(* CODESYS project Magazijn Structured Tekst 2V0 - Opdracht 3.project
   Company: Avans
   Description: Simulatie voor opstelling Sorteer Station.
   Title: Simulatie Sorteer Station
   Author: Rene Potters/Gerard Harkema
   Version: 0.1.0

Project tree, tasks and I/O mapping:
  Device : CODESYS Control Win V3, 3S - Smart Software Solutions GmbH, version 3.5.13.20
    application MagazijnOverzetterStation
      libraries: Standard, * (System); Util, * (System); VisuDialogs, 3.5.12.0 (System)
      task MainTask (cyclic, interval t#20ms, priority 1) calls Main
      task Simulatie (cyclic, interval t#20ms, priority 1) calls OverzetterSim, MagazijnSim
    application MagazijnTest
      libraries: Standard, * (System); Util, * (System); VisuDialogs, 3.5.12.0 (System)
      task MainTask (cyclic, interval t#20ms, priority 1) calls MagazijnTest
      task Simulatie (cyclic, interval t#20ms, priority 1) calls MagazijnSim
    application OverzetterTest
      libraries: Standard, * (System); Util, * (System); VisuDialogs, 3.5.12.0 (System)
      task MainTask (cyclic, interval t#20ms, priority 1) calls OverzetterTest
      task Simulatie (cyclic, interval t#20ms, priority 1) calls OverzetterSim
  Simulatie/
    program MagazijnSim [ST]
    global variables SIM
    program OverzetterSim [ST]
    data type OverzetterDUT
    data type MagazijnDUT
  text list GlobalTextList
  Programma Structured Text/
    function block OverzetterClass [ST]
    function block MagazijnClass [ST]
    program Main [ST]
    function block MagazijnOverzetterClass [ST]: initialize, cycle
    TestProgramms/
      program MagazijnTest [ST]
      program OverzetterTest [ST]
    States/
      data type magazijnStates
      data type magazijnOverzetterStationStates
  global variables GVL
  Visualisaties/
    visualisation MagazijnOverzetterStationHMI
    visualisation BekerMagazijnHMI
    visualisation OverzetterHMI
*)

// Simulatie/OverzetterDUT
{attribute 'qualified_only'}
{attribute 'strict'}
TYPE OverzetterDUT :
(
	INHETMIDDEN, NAARRECHTS, ISRECHTS, NAARLINKS, ISLINKS, GEVALLEN
);
END_TYPE

// Simulatie/MagazijnDUT
{attribute 'qualified_only'}
{attribute 'strict'}
TYPE MagazijnDUT :
(
	INGETROKKEN, INTREKKEN, UITGESTOTEN, UITSTOTEN, LEEG
);
END_TYPE

// Programma Structured Text/States/magazijnStates
// Datum : 17 december 2020, Auteur: Gerard Harkema
{attribute 'qualified_only'}
{attribute 'strict'}
TYPE magazijnStates :
(
	idle := 0,
	in,
	travel_out,
	out,
	travel_in,
	error
);
END_TYPE

// Programma Structured Text/States/magazijnOverzetterStationStates
// Datum : 17 december 2020, Auteur: Gerard Harkema
{attribute 'qualified_only'}
{attribute 'strict'}
TYPE magazijnOverzetterStationStates :
(
	idle := 0,
	wacht_op_klaar,
	wacht_enable,
	product_uitgifte,
	product_overzetten,
	service,
	error
);
END_TYPE

// Simulatie/SIM
{attribute 'qualified_only'}
VAR_GLOBAL
	// Rotatie van de overzetter
	Vx_OvzRotate: INT := 0;
	// Visualisatie invisible blok
	Vx_OvzBlokLinks: BOOL := FALSE;
	// Visualisatie invisible blok
	Vx_OvzBlokOverzetter: BOOL := FALSE;
	// Visualisatie invisible blok
	Vx_OvzBlokRechts: BOOL := FALSE;
	// Visualisatie invisible blok
	Vx_OvzBlokGevallen: BOOL := FALSE;	
	// Magazijn opnieuw vullen (simulatie)
	Ix_MagazijnVullen 	: BOOL;
	// Goten legen (symulatie)
	Ix_GotenLegen	  	: BOOL;
	
	
	
	
	
	
	
	
	
	
	
	
	
	
	
	
	
	
	
	
	
	
	
	
	
	
	
	
	
	
	
	
	
	
	
	
	
	
	
	
	
	
	
	
	
	
	
	
	// Simulatie visualisatie 
	Vw_Rotate45: INT := 45;
	// Visualisatie X positie van de uitstoter
	Vw_MagUitstoterBekerX: INT := 30;
	// Visualisatie invisible blok uitgestoten
	Vx_MagBlokUit: BOOL := TRUE;
	// Visualisatie invisible blok 1
	Vx_MagBlok1: BOOL := TRUE;
	// Visualisatie invisible blok 2
	Vx_MagBlok2: BOOL := TRUE;
	// Visualisatie invisible blok 3
	Vx_MagBlok3: BOOL := TRUE;
	// Visualisatie invisible blok 4
	Vx_MagBlok4: BOOL := TRUE;
	// Visualisatie invisible blokken
	Vx_MagBlok: ARRAY[1..8] OF BOOL;
	// Aantal blokken in het magazijn
	Vw_MagBlokAantal: INT := 4;
	// Simulatie onthoudt dat een blok maar 1x wordt uitgestoten
	Vw_MagBlok1X: INT := 0;
	// Ligt er een blok op band
	Vw_SorBlokBand: BOOL := FALSE;
	// Rotatie van de stopper
	Vw_SorStopperRotate: INT := 0;
	// Rotatie van de stopper goot 1
	Vw_SorGoot1Rotate: INT := 0;
	// Rotatie van de stopper goot 2
	Vw_SorGoot2Rotate: INT := 0;
	// Kleur van de blok op betreffende positie
	Vw_SorKleurBand: DWORD := 0;
	// Bewegen van de blok over de band
	Vi_SorBlokBandX: INT := 0;
	// Bewegen van de blok over de band
	Vi_SorBlokBandY: INT := 0;
	// Simulatie error. Inverse logica.
	Vx_MagLuchtDrukError: BOOL := TRUE;
	// Simulatie error. Inverse logica.
	Vx_MagIsInError: BOOL := TRUE;
	// Simulatie error. Inverse logica.
	Vx_MagIsUitError: BOOL := TRUE;
	// Simulatie error. Inverse logica.
	Vx_OvzLuchtDrukError: BOOL := TRUE;
	// Simulatie error. Inverse logica.
	Vx_OvzIsLinksError: BOOL := TRUE;
	// Simulatie error. Inverse logica.
	Vx_OvzIsRechtsError: BOOL := TRUE;
	// Simulatie error. Inverse logica.
	Vx_OvzVacuumError: BOOL := TRUE;
	// Simulatie error. Inverse logica.
	Vx_SorMotorAfvoerError: BOOL := TRUE;
	// Simulatie error. Inverse logica.
	Vx_SorGoot1InError: BOOL := TRUE;
	// Simulatie error. Inverse logica.
	Vx_SorGoot1UitError: BOOL := TRUE;
	// Simulatie error. Inverse logica.
	Vx_SorInGootError: BOOL := TRUE;
	// Ligt er een blok op de betreffende positie
	Vx_SorBlokGoot: ARRAY [1..3,1..6] OF BOOL;
	// Kleur van de blok op betreffende positie
	Vw_SorKleurGoot: ARRAY [1..3,1..6] OF DWORD;
END_VAR

// GVL
VAR_GLOBAL
	// Indrukken resetknop 
	Ix_Resetknop: BOOL;
	// Keuzeknop staat op hand
	Ix_Hand: BOOL;
	// Keuzeknop staat op auto
	Ix_Auto: BOOL;
	// Indrukken noodstop
	Ix_Noodstop: BOOL;
	// Bekers magazijn zijn op
	Ix_MagazijnLeeg: BOOL;
	// Beker is uit dekselmagazijn gestoten
	Ix_UitstoterBekerIn: BOOL;
	// Uitstoter Beker haalt nieuwe beker op
	Ix_UitstoterBekerUit: BOOL;
	// Indrukken startknop
	Ix_Stopknop: BOOL := TRUE;
	// Indrukken stopknop
	Ix_Startknop: BOOL;	
	//Perslucht is aanwezig
	Ix_PersluchtAanwezig :BOOL;
	//Werkstuk door overzetter opgepakt
	Ix_VacuumAanwezig :BOOL;
	//Overzetter haalt beker op(linker pos.)
	Ix_OverzetterIsLinks :BOOL;
	//Overzetter plaatst beker op sorteerpositie
	Ix_OverzetterIsRechts :BOOL;
	//Beker aanwezig op detectiepositie
	Ix_BekerAanwezig :BOOL;
	//Beker is van aluminium
	Ix_BekerMetaal :BOOL;
	//Beker reflecteert en is dus niet zwart
	Ix_BekerReflecteerd :BOOL;
	//Product is naar een van de goten gegaan
	Ix_BekerInGoot :BOOL;
	//Pusher uitvoergoot 1 is in
	Ix_UitvoerGoot1IsIn :BOOL;
	//Pusher uitvoergoot 2 is in
	Ix_UitvoerGoot2IsIn :BOOL;
	//Beker afvoeren is bezig
	Ix_StationAfvoerVrij :BOOL;
	//Pusher uitvoergoot 1 is uit
	Ix_UitvoerGoot1IsUit :BOOL;
	//Pusher uitvoergoot 2 is uit
	Ix_UitvoerGoot2IsUit :BOOL;
	// Beker uit magazijn stoten
	Qx_BekerUitstoten: BOOL;	
	//Beker oppakken
	Qx_VacuumAan :BOOL;
	//Beker loslaten
	Qx_BekerLossen :BOOL;
	//Overzetter naar bekermagazijn
	Qx_OverzetterLinks :BOOL;
	//Overzetter naar sorteerpositie
	Qx_OverzetterRechts :BOOL;
	//Transportband aan
	Qx_MotorAfvoerAan :BOOL;
	//Pusher goot 1 uit
	Qx_UitvoerGoot1Uit :BOOL;
	//Pusher goot 2 uit
	Qx_UitvoerGoot2Uit :BOOL;
	//Beker stoppen op band voor detectie
	Qx_StopperUit :BOOL;
	//Uitsorteren is bezet
	Qx_StationBezet :BOOL;
	// Visualisatie invisible Gele vlak
	Qx_GeleLamp: BOOL;
	// Visualisatie invisible groene vlak
	Qx_GroeneLamp: BOOL;
	// Visualisatie invisible rode vlak
	Qx_RodeLamp: BOOL;
END_VAR

// Programma Structured Text/Main
// Datum : 17 december 2020, Auteur: Gerard Harkema
PROGRAM Main
VAR
	sorteerStation 		: MagazijnOverzetterClass;
	initialized 		: BOOL := FALSE;
END_VAR

IF NOT initialized THEN
	// Forse Persluct aanwezig
	Ix_PersluchtAanwezig := TRUE;

	sorteerStation.initialize();
	initialized := TRUE;
END_IF

sorteerStation.cycle();

END_PROGRAM

// Programma Structured Text/MagazijnOverzetterClass
// Datum : 17 december 2020, Auteur: Gerard Harkema
FUNCTION_BLOCK MagazijnOverzetterClass
VAR
	// ******** Magazijn ********/
	magazijn		: MagazijnClass;
	
	// ******** Overzetter ********/
	overzetter		: OverzetterClass;

	eState 			: magazijnOverzetterStationStates := magazijnOverzetterStationStates.idle;
	x_Klaar 	: BOOL := FALSE;
	x_Error 	: BOOL := FALSE;
	x_Enable 	: BOOL := FALSE;

END_VAR

// ******** Magazijn ********/
	
// ******** Overzetter ********/

// ******** Sorteergoot ********/

// Datum : 17 december 2020, Auteur: Gerard Harkema
METHOD initialize
VAR
	// ******** Magazijn ********/
	// Bekers magazijn zijn op
	Ix_MagazijnLeegRef			: REFERENCE TO BOOL;
	// Beker is uit dekselmagazijn gestoten
	Ix_UitstoterBekerInRef		: REFERENCE TO BOOL;
	// Uitstoter Beker haalt nieuwe beker op
	Ix_UitstoterBekerUitRef		: REFERENCE TO BOOL;
	// Beker uit magazijn stoten
	Qx_BekerUitstotenRef		: REFERENCE TO BOOL;

	// ******** Overzetter ********/
	//Werkstuk door overzetter opgepakt
	Ix_VacuumAanwezigRef 		:REFERENCE TO BOOL;
	//Overzetter haalt beker op(linker pos.)
	Ix_OverzetterIsLinksRef 	:REFERENCE TO BOOL;
	//Overzetter plaatst beker op sorteerpositie
	Ix_OverzetterIsRechtsRef 	:REFERENCE TO BOOL;
	//Beker aanwezig op detectiepositie
	
	//Beker oppakken
	Qx_VacuumAanRef 			:REFERENCE TO BOOL;
	//Beker loslaten
	Qx_BekerLossenRef 			:REFERENCE TO BOOL;
	//Overzetter naar bekermagazijn
	Qx_OverzetterLinksRef		:REFERENCE TO BOOL;
	//Overzetter naar sorteerpositie
	Qx_OverzetterRechtsRef 		:REFERENCE TO BOOL;
	
END_VAR
// ******** Magazijn ********/
Ix_MagazijnLeegRef 			REF= gvl.Ix_MagazijnLeeg;
Ix_UitstoterBekerInRef 		REF= gvl.Ix_UitstoterBekerIn;
Ix_UitstoterBekerUitRef 	REF= gvl.Ix_UitstoterBekerUit;
Qx_BekerUitstotenRef 		REF= gvl.Qx_BekerUitstoten;

magazijn.initialize(Ix_MagazijnLeegRef,
					Ix_UitstoterBekerInRef,
					Ix_UitstoterBekerUitRef,
					Qx_BekerUitstotenRef,
					Ix_PersluchtAanwezig);
						

// ******** Overzetter ********/
//Werkstuk door overzetter opgepakt
Ix_VacuumAanwezigRef 		REF= Ix_VacuumAanwezig;
//Overzetter haalt beker op(linker pos.)
Ix_OverzetterIsLinksRef 	REF= Ix_OverzetterIsLinks;
//Overzetter plaatst beker op sorteerpositie
Ix_OverzetterIsRechtsRef 	REF= Ix_OverzetterIsRechts;

	//Beker oppakken
Qx_VacuumAanRef 			REF= Qx_VacuumAan;
//Beker loslaten
Qx_BekerLossenRef 			REF= Qx_BekerLossen;
//Overzetter naar bekermagazijn
Qx_OverzetterLinksRef		REF= Qx_OverzetterLinks;
//Overzetter naar sorteerpositie
Qx_OverzetterRechtsRef 		REF= Qx_OverzetterRechts;
	
overzetter.initialize(Ix_VacuumAanwezigRef,
					  Ix_OverzetterIsLinksRef,
					  Ix_OverzetterIsRechtsRef,
					  Qx_VacuumAanRef,
					  Qx_BekerLossenRef,
					  Qx_OverzetterLinksRef,
					  Qx_OverzetterRechtsRef);
END_METHOD

// Datum : 17 december 2020, Auteur: Gerard Harkema
METHOD cycle
VAR

END_VAR
x_Klaar := magazijn.isKlaar() 
	   AND overzetter.isKlaar();

x_Error := magazijn.isError()
	   OR overzetter.isError();
	   
	   
IF x_Error THEN
	eState := magazijnOverzetterStationStates.error;
END_IF

IF Ix_Startknop THEN
	x_Enable := TRUE;
	Ix_Startknop := FALSE;
END_IF
	  
IF not Ix_Stopknop THEN
	x_Enable := FALSE;
END_IF

IF Ix_ResetKnop THEN
	magazijn.reset();
	overzetter.reset();
	x_Enable := FALSE;
	eState := magazijnOverzetterStationStates.wacht_op_klaar;
END_IF

IF Ix_Noodstop THEN
	magazijn.noodstop();
	overzetter.noodstop();
	eState := magazijnOverzetterStationStates.error;
END_IF

Qx_GroeneLamp	:= NOT x_Klaar;
Qx_RodeLamp 	:= x_Error;

 
CASE eState OF
	magazijnOverzetterStationStates.idle:
		eState := magazijnOverzetterStationStates.wacht_op_klaar;
	magazijnOverzetterStationStates.wacht_op_klaar:
		IF x_Klaar THEN
			eState := magazijnOverzetterStationStates.wacht_enable;
		END_IF
	magazijnOverzetterStationStates.wacht_enable:
		IF magazijn.isMagazijnLeeg() THEN
			Qx_GeleLamp		:= TRUE;
			eState := magazijnOverzetterStationStates.service;
		ELSE
			IF x_Enable THEN
				magazijn.start();
				eState := magazijnOverzetterStationStates.product_uitgifte;
			END_IF
		END_IF
	magazijnOverzetterStationStates.product_uitgifte:
		IF magazijn.isKlaar() THEN
			overzetter.start();
			eState := magazijnOverzetterStationStates.product_overzetten;
		END_IF
	magazijnOverzetterStationStates.product_overzetten:
		IF overzetter.isKlaar() THEN
			eState := magazijnOverzetterStationStates.wacht_enable;
		END_IF
	magazijnOverzetterStationStates.service:
		IF Ix_Startknop THEN
			Qx_GeleLamp		:= FALSE;
			eState := magazijnOverzetterStationStates.wacht_enable;
		END_IF

END_CASE;


magazijn.cycle();
overzetter.cycle();
END_METHOD

END_FUNCTION_BLOCK

// Programma Structured Text/MagazijnClass
// Datum : 17 december 2020, Auteur: Gerard Harkema
FUNCTION_BLOCK MagazijnClass
VAR
	xInitialized				: BOOL := FALSE;
	
END_VAR

IF NOT xInitialized THEN

	xInitialized				:= TRUE;

END_IF

END_FUNCTION_BLOCK

// Programma Structured Text/OverzetterClass
// Datum : 17 december 2020, Auteur: Gerard Harkema
FUNCTION_BLOCK OverzetterClass
VAR
	xInitialized				: BOOL := FALSE;
END_VAR

IF NOT xInitialized THEN

	xInitialized				:= TRUE;

END_IF

END_FUNCTION_BLOCK

// Simulatie/OverzetterSim
PROGRAM OverzetterSim
VAR
	// Timer om overzetten te vertragen
	Fb_Pulse: BLINK;
	// Timer om overzetten te vertragen
	Fb_Trigger: F_TRIG;
	// Eerste keer om visualisatie te updaten
	Mx_FirstTime: BOOL := TRUE;
	// Afhandeling van de overzetter
	Me_OvzState: OverzetterDUT := OVERZETTERDUT.INHETMIDDEN;	
	// Afhandeling van het blokje
	Me_BlokState: OverzetterDUT := OVERZETTERDUT.INHETMIDDEN;	
	// Duurt even voor het vacuum aanwezig is
	Mi_VacuumCntr: INT := 0;	
END_VAR
VAR CONSTANT


	// Inverse logica
	INVISABLE: BOOL := TRUE;
	// Inverse logica
	VISABLE: BOOL := FALSE;

END_VAR

// Initialisatie.

IF (Mx_FirstTime) THEN
	Me_OvzState := OVERZETTERDUT.INHETMIDDEN;
	Me_BlokState := OVERZETTERDUT.ISLINKS;
	
	Mi_VacuumCntr := 0;
	SIM.Vx_OvzRotate := 0;
	Mx_FirstTime := FALSE;
END_IF

//
// Afhandelen van de pulse events. Hierdoor loopt de simulatie los van de 
// TASK tijd.
//
Fb_Pulse(ENABLE:=TRUE,TIMELOW:=T#100MS, TIMEHIGH:=T#100MS);
Fb_Trigger(CLK:=Fb_Pulse.OUT);


//
// Only if no emergency active, start handling the simulation.
//
IF (GVL.Ix_Noodstop) THEN
	Mx_FirstTime := TRUE;	
	RETURN;
END_IF
	
//
// The pulse determines the speed of the cilinder to move in
// ore move out. The cilinder is only moved if the airpressure 
// is available.
//
IF (Fb_Trigger.Q AND SIM.Vx_OvzLuchtDrukError) THEN
	
	//
	// De status van de arm wordt los afgehandeld van het blokje. De beweging
	// van de arm staat hier namelijk helemaal los van.
	//
	
	CASE Me_OvzState OF
		
		OVERZETTERDUT.INHETMIDDEN:
			// 
			// De arm is in beweging naar links of naar rechts.
			// Indien de arm in de uiterste positie is wordt er van 
			// state gewisseld. Aangezien de arm in beweging is staan
			// de eindschakelaars uit.
			//
			
			IF (GVL.Qx_OverzetterLinks) THEN
				IF (SIM.Vx_OvzRotate > -90) THEN
					GVL.Ix_OverzetterIsLinks := FALSE;	
					GVL.Ix_OverzetterIsRechts := FALSE;			
					SIM.Vx_OvzRotate := SIM.Vx_OvzRotate - 10;
				ELSE
					Me_OvzState := OVERZETTERDUT.ISLINKS;			
				END_IF	
				
			END_IF
				 
			IF (GVL.Qx_OverzetterRechts) THEN
				IF (SIM.Vx_OvzRotate < 90) THEN
					GVL.Ix_OverzetterIsLinks := FALSE;	
					GVL.Ix_OverzetterIsRechts := FALSE;				
					SIM.Vx_OvzRotate := SIM.Vx_OvzRotate + 10;
				ELSE
					Me_OvzState := OVERZETTERDUT.ISRECHTS;				
				END_IF			
			END_IF
				
		OVERZETTERDUT.ISLINKS:
		    //
			// Arm staat in een uiterste stand. Eindschakelaar is ingeschakeld.
			// Zodra de arm weer wordt bewogen verandert de state.
			//
			
			GVL.Ix_OverzetterIsLinks := TRUE AND SIM.Vx_OvzIsLinksError;	

			IF (GVL.Qx_OverzetterRechts AND NOT GVL.Qx_OverzetterLinks) THEN
				GVL.Ix_OverzetterIsLinks := FALSE;				
				Me_OvzState := OVERZETTERDUT.INHETMIDDEN;		
			END_IF
			
		OVERZETTERDUT.ISRECHTS:
		    //
			// Arm staat in een uiterste stand. Eindschakelaar is ingeschakeld.
			// Zodra de arm weer wordt bewogen verandert de state.
			//
		
			GVL.Ix_OverzetterIsRechts := TRUE AND SIM.Vx_OvzIsRechtsError;	

			IF (GVL.Qx_OverzetterLinks AND NOT GVL.Qx_OverzetterRechts) THEN
				GVL.Ix_OverzetterIsRechts := FALSE;				
				Me_OvzState := OVERZETTERDUT.INHETMIDDEN;		
			END_IF			
			
		END_CASE

	END_IF	

	//
	// De status van het blokje hangt af van een aantal stuursignalen zoals waar
	// de arm zich bevindt, of er vacuum is en of er een beker lossen wordt gegeven.
	//
	
	CASE Me_BlokState OF
		OVERZETTERDUT.ISLINKS:
			//
			// Als de arm links is moet er eerste een vacuum opgebouwd worden alvorens het blokje 
			// opgepakt kan worden. Daarna verandert de state. 
			//
			
			SIM.Vx_OvzBlokGevallen 	 := INVISABLE;
			SIM.Vx_OvzBlokLinks 	 := VISABLE;
			SIM.Vx_OvzBlokOverzetter := INVISABLE;
			SIM.Vx_OvzBlokRechts 	 := INVISABLE;
			
			IF (GVL.Qx_VacuumAan AND SIM.Vx_OvzVacuumError AND GVL.Ix_OverzetterIsLinks) AND (NOT GVL.Qx_BekerLossen) THEN
				Mi_VacuumCntr := Mi_VacuumCntr + 1;
			END_IF
			
			IF (NOT GVL.Qx_VacuumAan AND SIM.Vx_OvzVacuumError) THEN
				Mi_VacuumCntr := 0;
			END_IF

			GVL.Ix_VacuumAanwezig := (Mi_VacuumCntr > 50);
	
			IF  ( GVL.Ix_VacuumAanwezig AND (Me_OvzState = OVERZETTERDUT.INHETMIDDEN)) THEN
				Me_BlokState := OVERZETTERDUT.INHETMIDDEN;
			END_IF
			
		OVERZETTERDUT.INHETMIDDEN:
			//
			// Het blokje is in beweging zolang er vacuum is. Als er geen vacuum meer is
			// valt het blokje... Indien de arm helemaal rechts is kan het blokje gelost 
			// worden. Dit moet met een Bekerlossen ondanks het feit dat er
			// geen vacuum meer is....
			//
			
			SIM.Vx_OvzBlokGevallen 	 := INVISABLE;
			SIM.Vx_OvzBlokLinks 	 := INVISABLE;
			SIM.Vx_OvzBlokOverzetter := VISABLE;
			SIM.Vx_OvzBlokRechts 	 := INVISABLE;

		 	IF (GVL.Ix_OverzetterIsRechts) AND (NOT GVL.Qx_VacuumAan) AND (GVL.Qx_BekerLossen) THEN
				GVL.Ix_VacuumAanwezig := FALSE;
				Me_BlokState := OVERZETTERDUT.ISRECHTS;		
				RETURN;		
			END_IF
			
			IF (NOT GVL.Ix_OverzetterIsRechts) AND (NOT GVL.Ix_OverzetterIsLinks) AND(NOT GVL.Qx_VacuumAan) THEN
				GVL.Ix_VacuumAanwezig := FALSE;
				Me_BlokState := OVERZETTERDUT.GEVALLEN;				
			END_IF

		OVERZETTERDUT.ISRECHTS:	
		    // 
			// Blokje is gelost. Nu is het wachten tot de overzetter terug naar links wordt gestuurd. Daarna verdwijnt
			// het blokje automatisch.
			//
			
			SIM.Vx_OvzBlokGevallen 	 := INVISABLE;
			SIM.Vx_OvzBlokLinks 	 := INVISABLE;
			SIM.Vx_OvzBlokOverzetter := INVISABLE;
			SIM.Vx_OvzBlokRechts 	 := VISABLE;
			
			IF (NOT GVL.Ix_OverzetterIsRechts) THEN
				Me_BlokState := OVERZETTERDUT.ISLINKS;					
			END_IF

		OVERZETTERDUT.GEVALLEN:
			//
			// Blokje is gevallen..... Situatie herstelt zich zodra de arm helemaal links staat.
			//
				
			SIM.Vx_OvzBlokGevallen 	 := VISABLE;
			SIM.Vx_OvzBlokLinks 	 := INVISABLE;
			SIM.Vx_OvzBlokOverzetter := INVISABLE;
			SIM.Vx_OvzBlokRechts 	 := INVISABLE;
			
			IF (GVL.Ix_OverzetterIsLinks) THEN
				Me_BlokState := OVERZETTERDUT.ISLINKS;					
			END_IF				
	END_CASE

END_PROGRAM

// Simulatie/MagazijnSim
PROGRAM MagazijnSim
VAR
	// Timer om uitstoten en intrekken te vertragen
	Fb_Pulse: BLINK;
	// Timer om intrekken te vertragen
	Fb_Trigger: F_TRIG;
	// Eerste keer om visualisatie te updaten
	Mx_FirstTime: BOOL := TRUE;
	// Afhandeling van het magazijn
	Me_MagState: MAGAZIJNDUT := MAGAZIJNDUT.INGETROKKEN;
END_VAR

//
// Common stuff.
//

IF (Mx_FirstTime) THEN
	SIM.Vw_MagBlokAantal := 8;
	SIM.Vx_MagBlokUit:= FALSE;
	
	Mx_FirstTime := FALSE;
END_IF

					
//
// Handle all pulse and trigger events.
//
Fb_Pulse(ENABLE:=TRUE,TIMELOW:=T#200MS, TIMEHIGH:=T#200MS);
Fb_Trigger(CLK:=Fb_Pulse.OUT);


//
// Only if no emergency active, start handling the simulation.
//
IF (SIM.Ix_MagazijnVullen) THEN
	Mx_FirstTime := TRUE;
	SIM.Ix_MagazijnVullen := FALSE;
	RETURN;
END_IF
	
//
// The pulse determines the speed of the cilinder to move in
// ore move out. The cilinder is only moved if the airpressure 
// is available.
//
IF (Fb_Trigger.Q AND SIM.Vx_MagLuchtDrukError) THEN
		
			
	CASE Me_MagState OF
		MAGAZIJNDUT.INGETROKKEN:
			IF (SIM.Vx_MagBlokUit) THEN
				SIM.Vw_MagBlokAantal := SIM.Vw_MagBlokAantal - 1;
			END_IF
		
			SIM.Vw_MagUitstoterBekerX := 1;
			SIM.Vw_MagBlok1X    	  := SIM.Vw_MagUitstoterBekerX;
			SIM.Vx_MagBlokUit         := FALSE;
	
			IF (Qx_BekerUitstoten) THEN
				Me_MagState := MAGAZIJNDUT.UITSTOTEN;
			END_IF

		MAGAZIJNDUT.INTREKKEN:
			SIM.Vw_MagUitstoterBekerX := SIM.Vw_MagUitstoterBekerX - 30;
			
			IF (SIM.Vw_MagUitstoterBekerX < 0) THEN 
				SIM.Vw_MagUitstoterBekerX := 0; 
			END_IF		
			
			IF (SIM.Vw_MagUitstoterBekerX = 0) THEN
				Me_MagState := MAGAZIJNDUT.INGETROKKEN;				
			END_IF		

			IF (Qx_BekerUitstoten) THEN
				Me_MagState := MAGAZIJNDUT.UITSTOTEN;
			END_IF	
	
		MAGAZIJNDUT.UITGESTOTEN:
			SIM.Vx_MagBlokUit         := SIM.Vx_MagBlok1;
						
			IF (NOT Qx_BekerUitstoten) THEN
				Me_MagState := MAGAZIJNDUT.INTREKKEN;
			END_IF	
		
		MAGAZIJNDUT.UITSTOTEN:
			SIM.Vw_MagUitstoterBekerX := SIM.Vw_MagUitstoterBekerX + 30;
			SIM.Vw_MagBlok1X    	  := SIM.Vw_MagUitstoterBekerX;			
		
			IF (SIM.Vw_MagUitstoterBekerX > 70) THEN
				Me_MagState := MAGAZIJNDUT.UITGESTOTEN;				
			END_IF		

			IF (NOT Qx_BekerUitstoten) THEN
				Me_MagState := MAGAZIJNDUT.INTREKKEN;
			END_IF	
		
	END_CASE

	GVL.Ix_UitstoterBekerIn  := (Me_MagState = MAGAZIJNDUT.INGETROKKEN) AND SIM.Vx_MagIsInError;
	GVL.Ix_UitstoterBekerUit := (Me_MagState = MAGAZIJNDUT.UITGESTOTEN) AND SIM.Vx_MagIsUitError;	
	GVL.Ix_MagazijnLeeg 	 := (SIM.Vw_MagBlokAantal <= 0) AND (Ix_UitstoterBekerIn);	
	
	SIM.Vx_MagBlok[8] := (SIM.Vw_MagBlokAantal >= 8);
	SIM.Vx_MagBlok[7] := (SIM.Vw_MagBlokAantal >= 7);
	SIM.Vx_MagBlok[6] := (SIM.Vw_MagBlokAantal >= 6);
	SIM.Vx_MagBlok[5] := (SIM.Vw_MagBlokAantal >= 5);		
	SIM.Vx_MagBlok[4] := (SIM.Vw_MagBlokAantal >= 4);
	SIM.Vx_MagBlok[3] := (SIM.Vw_MagBlokAantal >= 3);
	SIM.Vx_MagBlok[2] := (SIM.Vw_MagBlokAantal >= 2);
	SIM.Vx_MagBlok[1] := (SIM.Vw_MagBlokAantal >= 1);	
	
END_IF

END_PROGRAM

// Programma Structured Text/TestProgramms/MagazijnTest
// Datum : 17 december 2020, Auteur: Gerard Harkema
PROGRAM MagazijnTest
VAR
	xInitialaized				: BOOL := FALSE;
	
	// Bekers magazijn zijn op
	Ix_MagazijnLeegRef			: REFERENCE TO BOOL;
	// Beker is uit dekselmagazijn gestoten
	Ix_UitstoterBekerInRef		: REFERENCE TO BOOL;
	// Uitstoter Beker haalt nieuwe beker op
	Ix_UitstoterBekerUitRef		: REFERENCE TO BOOL;
	// Beker uit magazijn stoten
	Qx_BekerUitstotenRef		: REFERENCE TO BOOL;
	
	magazijn: MagazijnClass;
	
END_VAR

IF NOT xInitialaized THEN

	// Forse Persluct aanwezig
	gvl.Ix_PersluchtAanwezig := TRUE;
	
	Ix_MagazijnLeegRef 			REF= gvl.Ix_MagazijnLeeg;
	Ix_UitstoterBekerInRef 		REF= gvl.Ix_UitstoterBekerIn;
	Ix_UitstoterBekerUitRef 	REF= gvl.Ix_UitstoterBekerUit;
	Qx_BekerUitstotenRef 		REF= gvl.Qx_BekerUitstoten;

	magazijn.initialize(Ix_MagazijnLeegRef,
					    Ix_UitstoterBekerInRef,
						Ix_UitstoterBekerUitRef,
						Qx_BekerUitstotenRef,
						Ix_PersluchtAanwezig);
	

	xInitialaized	:= TRUE;
END_IF

IF Ix_Startknop THEN
	magazijn.start();
	Ix_Startknop := FALSE;
END_IF

IF Ix_Resetknop THEN
	magazijn.reset();
END_IF

IF Ix_Noodstop THEN
	magazijn.noodstop();
END_IF

Qx_GroeneLamp := magazijn.isKlaar();
Qx_RodeLamp := magazijn.isError();
Qx_GeleLamp := magazijn.isMagazijnLeeg();
 
magazijn.cycle();

END_PROGRAM

// Programma Structured Text/TestProgramms/OverzetterTest
// Datum : 17 december 2020, Auteur: Gerard Harkema
PROGRAM OverzetterTest
VAR
	xInitialaized				: BOOL := FALSE;

	//Werkstuk door overzetter opgepakt
	Ix_VacuumAanwezigRef 		:REFERENCE TO BOOL;
	//Overzetter haalt beker op(linker pos.)
	Ix_OverzetterIsLinksRef 	:REFERENCE TO BOOL;
	//Overzetter plaatst beker op sorteerpositie
	Ix_OverzetterIsRechtsRef 	:REFERENCE TO BOOL;
	//Beker aanwezig op detectiepositie
	
	//Beker oppakken
	Qx_VacuumAanRef 			:REFERENCE TO BOOL;
	//Beker loslaten
	Qx_BekerLossenRef 			:REFERENCE TO BOOL;
	//Overzetter naar bekermagazijn
	Qx_OverzetterLinksRef		:REFERENCE TO BOOL;
	//Overzetter naar sorteerpositie
	Qx_OverzetterRechtsRef 		:REFERENCE TO BOOL;
	

	overzetter: OverzetterClass;
	
END_VAR

IF NOT xInitialaized THEN

	// Forse Persluct aanwezig
	gvl.Ix_PersluchtAanwezig := TRUE;
	
	//Werkstuk door overzetter opgepakt
	Ix_VacuumAanwezigRef 		REF= Ix_VacuumAanwezig;
	//Overzetter haalt beker op(linker pos.)
	Ix_OverzetterIsLinksRef 	REF= Ix_OverzetterIsLinks;
	//Overzetter plaatst beker op sorteerpositie
	Ix_OverzetterIsRechtsRef 	REF= Ix_OverzetterIsRechts;
	//Beker aanwezig op detectiepositie
	
		//Beker oppakken
	Qx_VacuumAanRef 			REF= Qx_VacuumAan;
	//Beker loslaten
	Qx_BekerLossenRef 			REF= Qx_BekerLossen;
	//Overzetter naar bekermagazijn
	Qx_OverzetterLinksRef		REF= Qx_OverzetterLinks;
	//Overzetter naar sorteerpositie
	Qx_OverzetterRechtsRef 		REF= Qx_OverzetterRechts;
	
	

	overzetter.initialize(Ix_VacuumAanwezigRef,
					      Ix_OverzetterIsLinksRef,
						  Ix_OverzetterIsRechtsRef,
						  Qx_VacuumAanRef,
						  Qx_BekerLossenRef,
						  Qx_OverzetterLinksRef,
						  Qx_OverzetterRechtsRef);
	

	xInitialaized	:= TRUE;
END_IF

IF Ix_Startknop THEN
	overzetter.start();
	Ix_Startknop := FALSE;
END_IF

IF Ix_Noodstop THEN
	overzetter.noodstop();
END_IF

IF Ix_Resetknop THEN
	overzetter.reset();
END_IF

Qx_GroeneLamp := overzetter.isKlaar();
Qx_RodeLamp := overzetter.isError();
 
overzetter.cycle();

END_PROGRAM

// Visualisaties/MagazijnOverzetterStationHMI
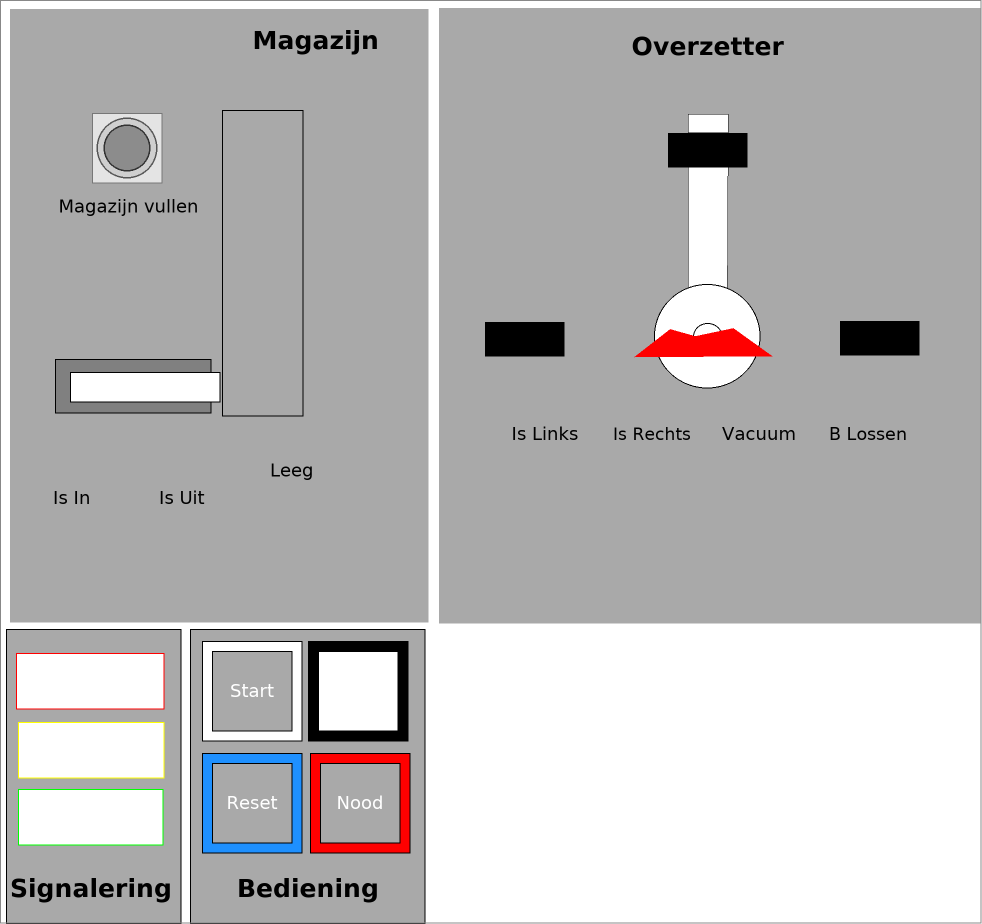
VISUALIZATION MagazijnOverzetterStationHMI  // 982x924
    Rectangle (9,8 420x615)
    Polygon (247,458) (277,458) (307,458) (337,458) (292,538), "Leeg", colour toggle: Ix_MagazijnLeeg
    Polygon (72,458) (72,458) (112,498) (72,538) (32,498), "Is In", colour toggle: Ix_UitstoterBekerIn
    Polygon (182,458) (182,458) (222,498) (182,538) (142,498), "Is Uit", colour toggle: Ix_UitstoterBekerUit
    Rectangle (55,359 156x54)
    Rectangle (222,110 81x306)
    Rectangle (314,373 61x29), colour toggle: SIM.Vx_MagBlokUit
    Rectangle (227,338 61x29), colour toggle: SIM.Vx_MagBlok[2]
    Rectangle (227,302 61x29), colour toggle: SIM.Vx_MagBlok[3]
    Rectangle (227,266 61x29), colour toggle: SIM.Vx_MagBlok[4]
    Rectangle (227,373 61x29), colour toggle: SIM.Vx_MagBlok[1]
        p3560616238: SIM.Vw_MagBlok1X
    Rectangle (70,372 150x30)
        p3560616238: SIM.Vw_MagUitstoterBekerX
    Label (241,25 150x30), "Magazijn"
    Group (6,629 175x295)
        Rectangle (0,0 175x295)
        Rectangle (10,24 148x56), colour toggle: Qx_RodeLamp
        Rectangle (12,93 146x56), colour toggle: Qx_GeleLamp
        Rectangle (12,160 145x56), colour toggle: Qx_GroeneLamp
        Label (10,236 150x46), "Signalering"
    Group (190,629 235x295)
        Rectangle (0,0 235x295)
        Group (12,12 100x100)
            RoundedRectangle (0,0 100x100)
            RoundedRectangle (10,10 80x80), "Start", tooltip "Start knop", colour toggle: Ix_Startknop
                OnMouseDown: execute { Ix_Startknop := TRUE; }
                OnMouseUp: execute { Ix_Startknop := FALSE; }
        Group (118,12 100x100)
            RoundedRectangle (0,0 100x100)
            RoundedRectangle (10,10 80x80), "Stop", tooltip "Stop knop", colour toggle: Ix_Stopknop
                OnMouseDown: execute { Ix_Stopknop := FALSE; }
                OnMouseUp: execute { Ix_Stopknop := TRUE; }
        Group (12,124 100x100)
            RoundedRectangle (0,0 100x100)
            RoundedRectangle (10,10 80x80), "Reset", tooltip "Reset knop", colour toggle: Ix_Resetknop
                OnMouseDown: execute { Ix_Resetknop := TRUE; }
                OnMouseUp: execute { Ix_Resetknop := FALSE; }
        Group (120,124 100x100)
            RoundedRectangle (0,0 100x100), "Nood"
            RoundedRectangle (10,10 80x80), "Nood", tooltip "Noodstop", colour toggle: Ix_Noodstop
                OnMouseDown: execute { Ix_Noodstop := NOT Ix_Noodstop; }
        Label (43,236 150x46), "Bediening"
    Group (6,629 175x295)
        Rectangle (0,0 175x295)
        Rectangle (10,24 148x56), colour toggle: Qx_RodeLamp
        Rectangle (12,93 146x56), colour toggle: Qx_GeleLamp
        Rectangle (12,160 145x56), colour toggle: Qx_GroeneLamp
        Label (10,236 150x46), "Signalering"
    Group (190,629 235x295)
        Rectangle (0,0 235x295)
        Group (12,12 100x100)
            RoundedRectangle (0,0 100x100)
            RoundedRectangle (10,10 80x80), "Start", tooltip "Start knop", colour toggle: Ix_Startknop
                OnMouseDown: execute { Ix_Startknop := TRUE; }
                OnMouseUp: execute { Ix_Startknop := FALSE; }
        Group (118,12 100x100)
            RoundedRectangle (0,0 100x100)
            RoundedRectangle (10,10 80x80), "Stop", tooltip "Stop knop", colour toggle: Ix_Stopknop
                OnMouseDown: execute { Ix_Stopknop := FALSE; }
                OnMouseUp: execute { Ix_Stopknop := TRUE; }
        Group (12,124 100x100)
            RoundedRectangle (0,0 100x100)
            RoundedRectangle (10,10 80x80), "Reset", tooltip "Reset knop", colour toggle: Ix_Resetknop
                OnMouseDown: execute { Ix_Resetknop := TRUE; }
                OnMouseUp: execute { Ix_Resetknop := FALSE; }
        Group (120,124 100x100)
            RoundedRectangle (0,0 100x100), "Nood"
            RoundedRectangle (10,10 80x80), "Nood", tooltip "Noodstop", colour toggle: Ix_Noodstop
                OnMouseDown: execute { Ix_Noodstop := NOT Ix_Noodstop; }
        Label (43,236 150x46), "Bediening"
    Group (6,629 175x295)
        Rectangle (0,0 175x295)
        Rectangle (10,24 148x56), colour toggle: Qx_RodeLamp
        Rectangle (12,93 146x56), colour toggle: Qx_GeleLamp
        Rectangle (12,160 145x56), colour toggle: Qx_GroeneLamp
        Label (10,236 150x46), "Signalering"
    Rectangle (6,629 175x295)
    Rectangle (16,653 148x56), colour toggle: Qx_RodeLamp
    Rectangle (18,722 146x56), colour toggle: Qx_GeleLamp
    Rectangle (18,789 145x56), colour toggle: Qx_GroeneLamp
    Label (16,865 150x46), "Signalering"
    Group (190,629 235x295)
        Rectangle (0,0 235x295)
        Group (12,12 100x100)
            RoundedRectangle (0,0 100x100)
            RoundedRectangle (10,10 80x80), "Start", tooltip "Start knop", colour toggle: Ix_Startknop
                OnMouseDown: execute { Ix_Startknop := TRUE; }
                OnMouseUp: execute { Ix_Startknop := FALSE; }
        Group (118,12 100x100)
            RoundedRectangle (0,0 100x100)
            RoundedRectangle (10,10 80x80), "Stop", tooltip "Stop knop", colour toggle: Ix_Stopknop
                OnMouseDown: execute { Ix_Stopknop := FALSE; }
                OnMouseUp: execute { Ix_Stopknop := TRUE; }
        Group (12,124 100x100)
            RoundedRectangle (0,0 100x100)
            RoundedRectangle (10,10 80x80), "Reset", tooltip "Reset knop", colour toggle: Ix_Resetknop
                OnMouseDown: execute { Ix_Resetknop := TRUE; }
                OnMouseUp: execute { Ix_Resetknop := FALSE; }
        Group (120,124 100x100)
            RoundedRectangle (0,0 100x100), "Nood"
            RoundedRectangle (10,10 80x80), "Nood", tooltip "Noodstop", colour toggle: Ix_Noodstop
                OnMouseDown: execute { Ix_Noodstop := NOT Ix_Noodstop; }
        Label (43,236 150x46), "Bediening"
    Rectangle (190,629 235x295)
    Group (202,641 100x100)
        RoundedRectangle (0,0 100x100)
        RoundedRectangle (10,10 80x80), "Start", tooltip "Start knop", colour toggle: Ix_Startknop
            OnMouseDown: execute { Ix_Startknop := TRUE; }
            OnMouseUp: execute { Ix_Startknop := FALSE; }
    RoundedRectangle (202,641 100x100)
    RoundedRectangle (212,651 80x80), "Start", tooltip "Start knop", colour toggle: Ix_Startknop
        OnMouseDown: execute { Ix_Startknop := TRUE; }
        OnMouseUp: execute { Ix_Startknop := FALSE; }
    Group (308,641 100x100)
        RoundedRectangle (0,0 100x100)
        RoundedRectangle (10,10 80x80), "Stop", tooltip "Stop knop", colour toggle: Ix_Stopknop
            OnMouseDown: execute { Ix_Stopknop := FALSE; }
            OnMouseUp: execute { Ix_Stopknop := TRUE; }
    RoundedRectangle (308,641 100x100)
    RoundedRectangle (318,651 80x80), "Stop", tooltip "Stop knop", colour toggle: Ix_Stopknop
        OnMouseDown: execute { Ix_Stopknop := FALSE; }
        OnMouseUp: execute { Ix_Stopknop := TRUE; }
    Group (202,753 100x100)
        RoundedRectangle (0,0 100x100)
        RoundedRectangle (10,10 80x80), "Reset", tooltip "Reset knop", colour toggle: Ix_Resetknop
            OnMouseDown: execute { Ix_Resetknop := TRUE; }
            OnMouseUp: execute { Ix_Resetknop := FALSE; }
    RoundedRectangle (202,753 100x100)
    RoundedRectangle (212,763 80x80), "Reset", tooltip "Reset knop", colour toggle: Ix_Resetknop
        OnMouseDown: execute { Ix_Resetknop := TRUE; }
        OnMouseUp: execute { Ix_Resetknop := FALSE; }
    Group (310,753 100x100)
        RoundedRectangle (0,0 100x100), "Nood"
        RoundedRectangle (10,10 80x80), "Nood", tooltip "Noodstop", colour toggle: Ix_Noodstop
            OnMouseDown: execute { Ix_Noodstop := NOT Ix_Noodstop; }
    RoundedRectangle (310,753 100x100), "Nood"
    RoundedRectangle (320,763 80x80), "Nood", tooltip "Noodstop", colour toggle: Ix_Noodstop
        OnMouseDown: execute { Ix_Noodstop := NOT Ix_Noodstop; }
    Label (233,865 150x46), "Bediening"
    Rectangle (227,194 61x29), colour toggle: SIM.Vx_MagBlok[6]
    Rectangle (227,158 61x29), colour toggle: SIM.Vx_MagBlok[7]
    Rectangle (227,122 61x29), colour toggle: SIM.Vx_MagBlok[8]
    Rectangle (227,229 61x29), colour toggle: SIM.Vx_MagBlok[5]
    Rectangle (438,7 544x617)
    Polygon (545,394) (545,394) (585,434) (545,474) (505,434), "Is Links", colour toggle: Ix_OverzetterisLinks
    Polygon (652,394) (652,394) (692,434) (652,474) (612,434), "Is Rechts", colour toggle: Ix_OverzetterIsRechts
    Polygon (759,394) (759,394) (799,434) (759,474) (719,434), "Vacuum", colour toggle: Ix_VacuumAanwezig
    Polygon (688,131) (703,131) (728,131) (727,310) (688,310)
        p2858320360: SIM.Vx_OvzRotate
    Polygon (868,394) (868,394) (908,434) (868,474) (828,434), "B Lossen", colour toggle: Qx_BekerLossen
    Polygon (688,114) (703,114) (728,114) (728,132) (688,132), colour toggle: Qx_VacuumAan
        p2858320360: SIM.Vx_OvzRotate
    Polygon (668,133) (683,133) (747,133) (747,167) (668,167), invisible if: SIM.Vx_OvzBlokOverzetter
        p2277200375: SIM.Vx_OvzRotate
    Polygon (485,322) (500,322) (564,322) (564,356) (485,356), invisible if: SIM.Vx_OvzBlokLinks
    Polygon (840,321) (855,321) (919,321) (919,355) (840,355), invisible if: SIM.Vx_OvzBlokRechts
    Ellipse (654,284 106x104)
    Ellipse (693,323 29x27)
    Polygon (670,329) (695,336) (733,328) (772,356) (634,357), invisible if: SIM.Vx_OvzBlokGevallen
        p2277200375: SIM.Vx_OvzRotate
    Label (606,31 204x30), "Overzetter"
    Polygon (51,194) (81,194) (111,194) (206,208) (106,222), "Magazijn vullen", colour toggle: Ix_MagazijnLeeg
    PushSwitch (92,113 70x70), tooltip "Magazijn vullen", variable: SIM.Ix_MagazijnVullen, behaviour: TOGGLE, style: Switch-PushSwitch-Gray
END_VISUALIZATION

// Visualisaties/BekerMagazijnHMI
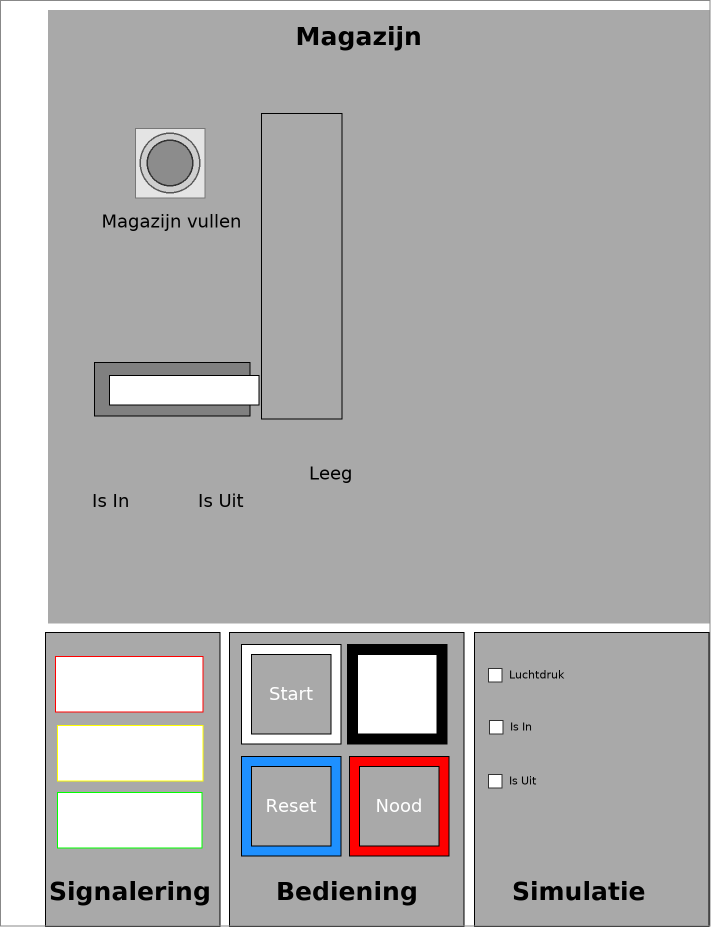
VISUALIZATION BekerMagazijnHMI  // 711x927
    Rectangle (47,9 664x615)
    Polygon (286,461) (316,461) (346,461) (376,461) (331,541), "Leeg", colour toggle: Ix_MagazijnLeeg
    Polygon (111,461) (111,461) (151,501) (111,541) (71,501), "Is In", colour toggle: Ix_UitstoterBekerIn
    Polygon (221,461) (221,461) (261,501) (221,541) (181,501), "Is Uit", colour toggle: Ix_UitstoterBekerUit
    Rectangle (94,362 156x54)
    Rectangle (261,113 81x306)
    Rectangle (353,376 61x29), colour toggle: SIM.Vx_MagBlokUit
    Rectangle (266,341 61x29), colour toggle: SIM.Vx_MagBlok[2]
    Rectangle (266,305 61x29), colour toggle: SIM.Vx_MagBlok[3]
    Rectangle (266,269 61x29), colour toggle: SIM.Vx_MagBlok[4]
    Rectangle (266,376 61x29), colour toggle: SIM.Vx_MagBlok[1]
        p3560616238: SIM.Vw_MagBlok1X
    Rectangle (109,375 150x30)
        p3560616238: SIM.Vw_MagUitstoterBekerX
    Label (284,21 150x30), "Magazijn"
    Group (45,632 664x295)
        Group (0,0 664x295)
            Group (429,0 235x295)
                Rectangle (0,0 235x295)
                Label (30,236 150x46), "Simulatie"
            Group (0,0 175x295)
                Rectangle (0,0 175x295)
                Rectangle (10,24 148x56), colour toggle: Qx_RodeLamp
                Rectangle (12,93 146x56), colour toggle: Qx_GeleLamp
                Rectangle (12,160 145x56), colour toggle: Qx_GroeneLamp
                Label (10,236 150x46), "Signalering"
            Group (184,0 235x295)
                Rectangle (0,0 235x295)
                Group (12,12 100x100)
                    RoundedRectangle (0,0 100x100)
                    RoundedRectangle (10,10 80x80), "Start", tooltip "Start knop", colour toggle: Ix_Startknop
                        OnMouseDown: execute { Ix_Startknop := TRUE; }
                        OnMouseUp: execute { Ix_Startknop := FALSE; }
                Group (118,12 100x100)
                    RoundedRectangle (0,0 100x100)
                    RoundedRectangle (10,10 80x80), "Stop", tooltip "Stop knop", colour toggle: Ix_Stopknop
                        OnMouseDown: execute { Ix_Stopknop := FALSE; }
                        OnMouseUp: execute { Ix_Stopknop := TRUE; }
                Group (12,124 100x100)
                    RoundedRectangle (0,0 100x100)
                    RoundedRectangle (10,10 80x80), "Reset", tooltip "Reset knop", colour toggle: Ix_Resetknop
                        OnMouseDown: execute { Ix_Resetknop := TRUE; }
                        OnMouseUp: execute { Ix_Resetknop := FALSE; }
                Group (120,124 100x100)
                    RoundedRectangle (0,0 100x100), "Nood"
                    RoundedRectangle (10,10 80x80), "Nood", tooltip "Noodstop", colour toggle: Ix_Noodstop
                        OnMouseDown: execute { Ix_Noodstop := NOT Ix_Noodstop; }
                Label (43,236 150x46), "Bediening"
        Checkbox (441,17 196x52), "Luchtdruk", variable: SIM.Vx_MagLuchtDrukError
        Checkbox (442,69 196x52), "Is In", variable: SIM.Vx_MagIsInError
        Checkbox (441,123 196x52), "Is Uit", variable: SIM.Vx_MagIsUitError
    Rectangle (266,197 61x29), colour toggle: SIM.Vx_MagBlok[6]
    Rectangle (266,161 61x29), colour toggle: SIM.Vx_MagBlok[7]
    Rectangle (266,125 61x29), colour toggle: SIM.Vx_MagBlok[8]
    Rectangle (266,232 61x29), colour toggle: SIM.Vx_MagBlok[5]
    PushSwitch (135,128 70x70), tooltip "Magazijn vullen", variable: SIM.Ix_MagazijnVullen, behaviour: TOGGLE, style: Switch-PushSwitch-Gray
    Polygon (94,209) (124,209) (154,209) (249,223) (149,237), "Magazijn vullen", colour toggle: Ix_MagazijnLeeg
END_VISUALIZATION

// Visualisaties/OverzetterHMI
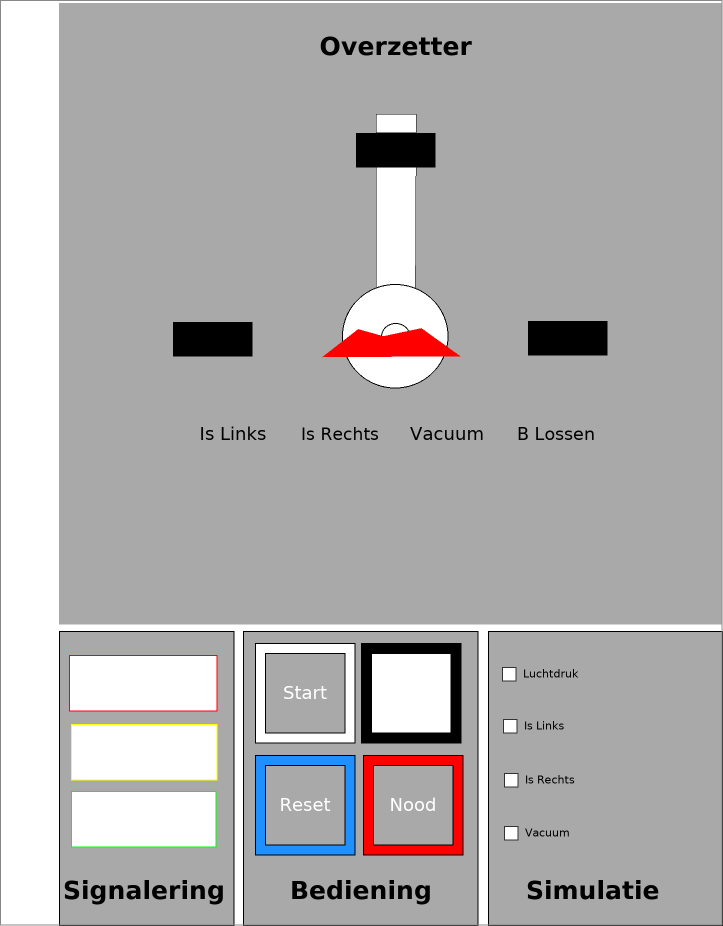
VISUALIZATION OverzetterHMI  // 723x926
    Rectangle (58,2 664x623)
    Polygon (233,394) (233,394) (273,434) (233,474) (193,434), "Is Links", colour toggle: Ix_OverzetterisLinks
    Polygon (340,394) (340,394) (380,434) (340,474) (300,434), "Is Rechts", colour toggle: Ix_OverzetterIsRechts
    Polygon (447,394) (447,394) (487,434) (447,474) (407,434), "Vacuum", colour toggle: Ix_VacuumAanwezig
    Polygon (376,131) (391,131) (416,131) (415,310) (376,310)
        p2858320360: SIM.Vx_OvzRotate
    Polygon (556,394) (556,394) (596,434) (556,474) (516,434), "B Lossen", colour toggle: Qx_BekerLossen
    Polygon (376,114) (391,114) (416,114) (416,132) (376,132), colour toggle: Qx_VacuumAan
        p2858320360: SIM.Vx_OvzRotate
    Polygon (356,133) (371,133) (435,133) (435,167) (356,167), invisible if: SIM.Vx_OvzBlokOverzetter
        p2277200375: SIM.Vx_OvzRotate
    Polygon (173,322) (188,322) (252,322) (252,356) (173,356), invisible if: SIM.Vx_OvzBlokLinks
    Polygon (528,321) (543,321) (607,321) (607,355) (528,355), invisible if: SIM.Vx_OvzBlokRechts
    Ellipse (342,284 106x104)
    Ellipse (381,323 29x27)
    Polygon (358,329) (383,336) (421,328) (460,356) (322,357), invisible if: SIM.Vx_OvzBlokGevallen
        p2277200375: SIM.Vx_OvzRotate
    Label (294,31 204x30), "Overzetter"
    Group (59,631 175x295)
        Rectangle (0,0 175x295)
        Rectangle (10,24 148x56), colour toggle: Qx_RodeLamp
        Rectangle (12,93 146x56), colour toggle: Qx_GeleLamp
        Rectangle (12,160 145x56), colour toggle: Qx_GroeneLamp
        Label (10,236 150x46), "Signalering"
    Group (243,631 235x295)
        Rectangle (0,0 235x295)
        Group (12,12 100x100)
            RoundedRectangle (0,0 100x100)
            RoundedRectangle (10,10 80x80), "Start", tooltip "Start knop", colour toggle: Ix_Startknop
                OnMouseDown: execute { Ix_Startknop := TRUE; }
                OnMouseUp: execute { Ix_Startknop := FALSE; }
        Group (118,12 100x100)
            RoundedRectangle (0,0 100x100)
            RoundedRectangle (10,10 80x80), "Stop", tooltip "Stop knop", colour toggle: Ix_Stopknop
                OnMouseDown: execute { Ix_Stopknop := FALSE; }
                OnMouseUp: execute { Ix_Stopknop := TRUE; }
        Group (12,124 100x100)
            RoundedRectangle (0,0 100x100)
            RoundedRectangle (10,10 80x80), "Reset", tooltip "Reset knop", colour toggle: Ix_Resetknop
                OnMouseDown: execute { Ix_Resetknop := TRUE; }
                OnMouseUp: execute { Ix_Resetknop := FALSE; }
        Group (120,124 100x100)
            RoundedRectangle (0,0 100x100), "Nood"
            RoundedRectangle (10,10 80x80), "Nood", tooltip "Noodstop", colour toggle: Ix_Noodstop
                OnMouseDown: execute { Ix_Noodstop := NOT Ix_Noodstop; }
        Label (43,236 150x46), "Bediening"
    Group (488,631 235x295)
        Group (0,0 235x295)
            Rectangle (0,0 235x295)
            Label (30,236 150x46), "Simulatie"
        Checkbox (12,17 196x52), "Luchtdruk", variable: SIM.Vx_OvzLuchtDrukError
        Checkbox (13,69 196x52), "Is Links", variable: SIM.Vx_OvzIsLinksError
        Checkbox (14,123 196x52), "Is Rechts", variable: SIM.Vx_OvzIsRechtsError
        Checkbox (14,176 196x52), "Vacuum", variable: SIM.Vx_OvzVacuumError
END_VISUALIZATION
